Fanuc KAREL source: kb00152.KL

-- PROVISIONAL review KL for V770-1; original PC SHA256 892ab83311b5fd1edb9ecb3c4d967e086141d6b44029d1ceb0f8e95cce23a9b6
-- Incomplete behavior may be omitted. Consult companion uncertainty JSON. Do not deploy.
PROGRAM KB00152
%NOLOCKGROUP
VAR
  P1 : REAL
  RESULT : INTEGER
BEGIN
  -- UNRESOLVED_PC offsets 5-16; opcodes 2E,23
  -- UNRESOLVED_PC offsets 21-36; opcodes 27,22,76,23
  -- UNRESOLVED_PC offsets 41-45; opcodes 7F
END KB00152
